{attribute 'GeneratedUsingTerminal: EJ7211-0011-0026'}
{attribute addProperty BoxType "EJ7211-0011-0026"}
{attribute addProperty Id "EtcSlaveTerminalBaseDS402_StatuswordAT %I*DS402_Statusword_9B36FDFC2DS402_Position_actual_valueAT %I*DS402_Position_actual_value_07DC4C744DS402_ControlwordAT %Q*DS402_Controlword_F3F147212DS402_Target_velocityAT %Q*DS402_Target_velocity_08A9583B4WcStateAT %I*WcState_9091E0EB2InfoDataAT %I*InfoData_96C94FAE19"}
{attribute addProperty CRC "731644075"}
{attribute addProperty Size "33"}
TYPE EJ7211_2B9C00AB EXTENDS EtcSlaveTerminalBase :
STRUCT
	{attribute addProperty Name "DS402_Statusword"}
	DS402_Statusword : DS402_Statusword_9B36FDFC;
	{attribute addProperty Name "DS402_Position_actual_value"}
	DS402_Position_actual_value : DS402_Position_actual_value_07DC4C74;
	{attribute addProperty Name "DS402_Controlword"}
	DS402_Controlword : DS402_Controlword_F3F14721;
	{attribute addProperty Name "DS402_Target_velocity"}
	DS402_Target_velocity : DS402_Target_velocity_08A9583B;
	{attribute addProperty Name "WcState"}
	WcState : WcState_9091E0EB;
	{attribute addProperty Name "InfoData"}
	InfoData : InfoData_96C94FAE;
END_STRUCT
END_TYPE

(* stored: Version 1.2.0.0, ProductVersion 3.1.4024.9
   DUT EJ7211_2B9C00AB: Id {bc780635-14ee-42aa-adb3-c3d7d2c6a40b} *)
